(* IEC 61131-3 sources: Lasal/CPU_5344_V01/Class/profileInfo, 1 file *)

(* ---- profileInfo.st ---- *)
(*!
<Class
	Name               = "profileInfo"
	Revision           = "0.0"
	RealtimeTask       = "false"
	CyclicTask         = "false"
	BackgroundTask     = "true"
	DefBackground      = "10 ms"
	Sigmatek           = "false"
	OSInterface        = "false"
	HighPriority       = "false"
	Automatic          = "false"
	UpdateMode         = "Prescan"
	SharedCommandTable = "true"
	Objectsize         = "(780,120)">
	<Channels>
		<Server Name="ClassSvr" Visualized="false" Initialize="false" WriteProtected="true" Retentive="false"/>
		<Server Name="length1" Visualized="true" Remotely="true" Initialize="false" WriteProtected="true" Retentive="false"/>
		<Server Name="length10" Visualized="true" Remotely="true" Initialize="false" WriteProtected="true" Retentive="false"/>
		<Server Name="length2" Visualized="true" Remotely="true" Initialize="false" WriteProtected="true" Retentive="false"/>
		<Server Name="length3" Visualized="true" Remotely="true" Initialize="false" WriteProtected="true" Retentive="false"/>
		<Server Name="length4" Visualized="true" Remotely="true" Initialize="false" WriteProtected="true" Retentive="false"/>
		<Server Name="length5" Visualized="true" Remotely="true" Initialize="false" WriteProtected="true" Retentive="false"/>
		<Server Name="length6" Visualized="true" Remotely="true" Initialize="false" WriteProtected="true" Retentive="false"/>
		<Server Name="length7" Visualized="true" Remotely="true" Initialize="false" WriteProtected="true" Retentive="false"/>
		<Server Name="length8" Visualized="true" Remotely="true" Initialize="false" WriteProtected="true" Retentive="false"/>
		<Server Name="length9" Visualized="true" Remotely="true" Initialize="false" WriteProtected="true" Retentive="false"/>
		<Server Name="recNr1" Visualized="true" Remotely="true" Initialize="false" WriteProtected="true" Retentive="false"/>
		<Server Name="recNr10" Visualized="true" Remotely="true" Initialize="false" WriteProtected="true" Retentive="false"/>
		<Server Name="recNr2" Visualized="true" Remotely="true" Initialize="false" WriteProtected="true" Retentive="false"/>
		<Server Name="recNr3" Visualized="true" Remotely="true" Initialize="false" WriteProtected="true" Retentive="false"/>
		<Server Name="recNr4" Visualized="true" Remotely="true" Initialize="false" WriteProtected="true" Retentive="false"/>
		<Server Name="recNr5" Visualized="true" Remotely="true" Initialize="false" WriteProtected="true" Retentive="false"/>
		<Server Name="recNr6" Visualized="true" Remotely="true" Initialize="false" WriteProtected="true" Retentive="false"/>
		<Server Name="recNr7" Visualized="true" Remotely="true" Initialize="false" WriteProtected="true" Retentive="false"/>
		<Server Name="recNr8" Visualized="true" Remotely="true" Initialize="false" WriteProtected="true" Retentive="false"/>
		<Server Name="recNr9" Visualized="true" Remotely="true" Initialize="false" WriteProtected="true" Retentive="false"/>
		<Client Name="ctrlAssemDb" Required="true" Internal="false"/>
		<Client Name="String1" Required="true" Internal="true"/>
		<Client Name="String10" Required="true" Internal="true"/>
		<Client Name="String2" Required="true" Internal="true"/>
		<Client Name="String3" Required="true" Internal="true"/>
		<Client Name="String4" Required="true" Internal="true"/>
		<Client Name="String5" Required="true" Internal="true"/>
		<Client Name="String6" Required="true" Internal="true"/>
		<Client Name="String7" Required="true" Internal="true"/>
		<Client Name="String8" Required="true" Internal="true"/>
		<Client Name="String9" Required="true" Internal="true"/>
	</Channels>
	<Network Name="profileInfo">
		<!-- List of Components in this network -->
		<Components>
			<Object
				Name       = "String1"
				Class      = "String"
				Position   = "(270,300)"
				Visualized = "true"
				Remotely   = "true">
				<Channels>
					<Server Name="Data"/>
					<Client Name="SingleRealloc" Value="1"/>
				</Channels>
			</Object>
			<Object
				Name       = "String10"
				Class      = "String"
				Position   = "(270,1650)"
				Visualized = "true"
				Remotely   = "true">
				<Channels>
					<Server Name="Data"/>
					<Client Name="SingleRealloc" Value="1"/>
				</Channels>
			</Object>
			<Object
				Name       = "String2"
				Class      = "String"
				Position   = "(270,450)"
				Visualized = "true"
				Remotely   = "true">
				<Channels>
					<Server Name="Data"/>
					<Client Name="SingleRealloc" Value="1"/>
				</Channels>
			</Object>
			<Object
				Name       = "String3"
				Class      = "String"
				Position   = "(270,600)"
				Visualized = "true"
				Remotely   = "true">
				<Channels>
					<Server Name="Data"/>
					<Client Name="SingleRealloc" Value="1"/>
				</Channels>
			</Object>
			<Object
				Name       = "String4"
				Class      = "String"
				Position   = "(270,750)"
				Visualized = "true"
				Remotely   = "true">
				<Channels>
					<Server Name="Data"/>
					<Client Name="SingleRealloc" Value="1"/>
				</Channels>
			</Object>
			<Object
				Name       = "String5"
				Class      = "String"
				Position   = "(270,900)"
				Visualized = "true"
				Remotely   = "true">
				<Channels>
					<Server Name="Data"/>
					<Client Name="SingleRealloc" Value="1"/>
				</Channels>
			</Object>
			<Object
				Name       = "String6"
				Class      = "String"
				Position   = "(270,1050)"
				Visualized = "true"
				Remotely   = "true">
				<Channels>
					<Server Name="Data"/>
					<Client Name="SingleRealloc" Value="1"/>
				</Channels>
			</Object>
			<Object
				Name       = "String7"
				Class      = "String"
				Position   = "(270,1200)"
				Visualized = "true"
				Remotely   = "true">
				<Channels>
					<Server Name="Data"/>
					<Client Name="SingleRealloc" Value="1"/>
				</Channels>
			</Object>
			<Object
				Name       = "String8"
				Class      = "String"
				Position   = "(270,1350)"
				Visualized = "true"
				Remotely   = "true">
				<Channels>
					<Server Name="Data"/>
					<Client Name="SingleRealloc" Value="1"/>
				</Channels>
			</Object>
			<Object
				Name       = "String9"
				Class      = "String"
				Position   = "(270,1500)"
				Visualized = "true"
				Remotely   = "true">
				<Channels>
					<Server Name="Data"/>
					<Client Name="SingleRealloc" Value="1"/>
				</Channels>
			</Object>
		</Components>
		<Comments>
		</Comments>
		<!-- List of Connections in this network -->
		<Connections>
			<Connection Source="this.String1" Destination="String1.Data"/>
			<Connection Source="this.String2" Destination="String2.Data"/>
			<Connection Source="this.String3" Destination="String3.Data"/>
			<Connection Source="this.String4" Destination="String4.Data"/>
			<Connection Source="this.String5" Destination="String5.Data"/>
			<Connection Source="this.String6" Destination="String6.Data"/>
			<Connection Source="this.String7" Destination="String7.Data"/>
			<Connection Source="this.String8" Destination="String8.Data"/>
			<Connection Source="this.String9" Destination="String9.Data"/>
			<Connection Source="this.String10" Destination="String10.Data"/>
		</Connections>
		<!-- Headerfiles -->
		<Options>
		</Options>
	</Network>
</Class>
*)
profileInfo : CLASS
	TYPE
#pragma pack(push, 1)
	  nameAndLength : STRUCT
	    name : gbl_datatypes::tStr20;
	    length : DINT;
	    recNr : DINT;
	  END_STRUCT;
#pragma pack(pop)
	END_TYPE
  //Servers:
	ClassSvr 	: SvrChCmd_DINT;
	length1 	: SvrCh_DINT;
	recNr1 	: SvrCh_DINT;
	length2 	: SvrCh_DINT;
	recNr2 	: SvrCh_DINT;
	length3 	: SvrCh_DINT;
	recNr3 	: SvrCh_DINT;
	length4 	: SvrCh_DINT;
	recNr4 	: SvrCh_DINT;
	length5 	: SvrCh_DINT;
	recNr5 	: SvrCh_DINT;
	length6 	: SvrCh_DINT;
	recNr6 	: SvrCh_DINT;
	length7 	: SvrCh_DINT;
	recNr7 	: SvrCh_DINT;
	length8 	: SvrCh_DINT;
	recNr8 	: SvrCh_DINT;
	length9 	: SvrCh_DINT;
	recNr9 	: SvrCh_DINT;
	length10 	: SvrCh_DINT;
	recNr10 	: SvrCh_DINT;
  //Clients:
	String1 	: CltChCmd_String;
	String2 	: CltChCmd_String;
	String3 	: CltChCmd_String;
	String4 	: CltChCmd_String;
	String5 	: CltChCmd_String;
	String6 	: CltChCmd_String;
	String7 	: CltChCmd_String;
	String8 	: CltChCmd_String;
	String9 	: CltChCmd_String;
	String10 	: CltChCmd_String;
	ctrlAssemDb 	: CltChCmd_AssemblyDbV2;
  //Variables:
		oldAmountDone 	: DINT;
		oldAmountToDo 	: DINT;
		oldRecepiNr 	: UDINT;
		cntr 	: DINT;
		cntr2 	: DINT;
		cntrRec 	: DINT;
		tmpAssembly 	: AssemblyDbV2::tRecipeData;
		initDone 	: DINT;
		strEmpty 	: gbl_datatypes::tStr20;
		data : ARRAY [1..10] OF nameAndLength;

		refreshCounter 	: DINT;
  //Functions:

	FUNCTION VIRTUAL GLOBAL Init;

	FUNCTION VIRTUAL GLOBAL Background
		VAR_INPUT
			EAX 	: UDINT;
		END_VAR
		VAR_OUTPUT
			state (EAX) 	: UDINT := READY;
		END_VAR;
  //Tables:
	FUNCTION @STD
		VAR_OUTPUT
			ret_code	: CONFSTATES;
		END_VAR;
	FUNCTION GLOBAL TAB @CT_;
END_CLASS;

#pragma using String
#pragma usingLtd AssemblyDbV2

// JdK 27-12-2019: profileInfo, set profile information of 10 next assemblies in string and length dints
// stop if one is already completed

FUNCTION VIRTUAL GLOBAL profileInfo::Background
	VAR_INPUT
		EAX 	: UDINT;
	END_VAR
	VAR_OUTPUT
		state (EAX) 	: UDINT;(* := READY *)
	END_VAR

  IF oldAmountDone <> ctrlAssemDb.AmountDone | oldAmountToDo <> ctrlAssemDb.AmountToDo |
        oldRecepiNr <> ctrlAssemDb.RecipeId | refreshCounter > 1000 THEN //on change, or after 10 seconds

    refreshCounter:= 0;
    oldAmountDone:= ctrlAssemDb.AmountDone;
    oldAmountToDo:= ctrlAssemDb.AmountToDo;
    oldRecepiNr:= ctrlAssemDb.RecipeId;
    cntrRec:=0;
    //first write all to empty
    FOR cntr:=1 TO 10 DO
      data[cntr].length:= 0;
      data[cntr].recNr:= 0;
      data[cntr].name:=strEmpty;
    END_FOR;

    FOR cntr:=1 TO 10 DO //try a maximum of 10 assembly's
      tmpAssembly:=ctrlAssemDb.GetRecipe(id:=to_dint(ctrlAssemDb.RecipeId)+cntrRec);
      IF tmpAssembly.amountToDo > tmpAssembly.amountDone THEN
        FOR cntr2:=1 TO tmpAssembly.amountToDo - tmpAssembly.amountDone DO
          data[cntr].name:=tmpAssembly.description;
          data[cntr].length:=tmpAssembly.inputLength;
          data[cntr].recNr:= to_dint(ctrlAssemDb.RecipeId)+cntrRec;
          cntr+=1;
          IF cntr > 10 THEN
            exit; //only fill 10 data sets
          END_IF;
        END_FOR;
        cntrRec+=1;
        cntr-= 1; //counting up is already done, and because we are in for loop it's done again
      ELSE
        exit; //stop if amount of one of the assemblies is reached
      END_IF;

    END_FOR;

    //now write data to servers
    String1.WriteDataOff(udLen:=20, udOff:=0, pData:=#data[1].name[0]);  //.SetDataAt(pData:=#data[1].name[0], udAt:=0);
    String2.WriteDataOff(udLen:=20, udOff:=0, pData:=#data[2].name[0]);
    String3.WriteDataOff(udLen:=20, udOff:=0, pData:=#data[3].name[0]);
    String4.WriteDataOff(udLen:=20, udOff:=0, pData:=#data[4].name[0]);
    String5.WriteDataOff(udLen:=20, udOff:=0, pData:=#data[5].name[0]);
    String6.WriteDataOff(udLen:=20, udOff:=0, pData:=#data[6].name[0]);
    String7.WriteDataOff(udLen:=20, udOff:=0, pData:=#data[7].name[0]);
    String8.WriteDataOff(udLen:=20, udOff:=0, pData:=#data[8].name[0]);
    String9.WriteDataOff(udLen:=20, udOff:=0, pData:=#data[9].name[0]);
    String10.WriteDataOff(udLen:=20, udOff:=0, pData:=#data[10].name[0]);
    length1:=data[1].length;
    length2:=data[2].length;
    length3:=data[3].length;
    length4:=data[4].length;
    length5:=data[5].length;
    length6:=data[6].length;
    length7:=data[7].length;
    length8:=data[8].length;
    length9:=data[9].length;
    length10:=data[10].length;
    recNr1:=data[1].recNr;
    recNr2:=data[2].recNr;
    recNr3:=data[3].recNr;
    recNr4:=data[4].recNr;
    recNr5:=data[5].recNr;
    recNr6:=data[6].recNr;
    recNr7:=data[7].recNr;
    recNr8:=data[8].recNr;
    recNr9:=data[9].recNr;
    recNr10:=data[10].recNr;
  ELSE
    refreshCounter+= 1;
  END_IF;

END_FUNCTION

FUNCTION VIRTUAL GLOBAL profileInfo::Init

  IF initDone= 0 THEN
    _memset(dest:=#strEmpty[0], usByte:=0, cntr:=SIZEOF(strEmpty));
    _memcpy(ptr1:=#strEmpty[0], ptr2:="empty", cntr:=5);
    initDone:= 1;

  END_IF;

END_FUNCTION
